ABB RobotStudio station: Estacion2.rsstn

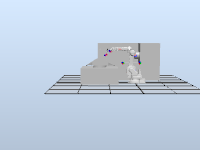
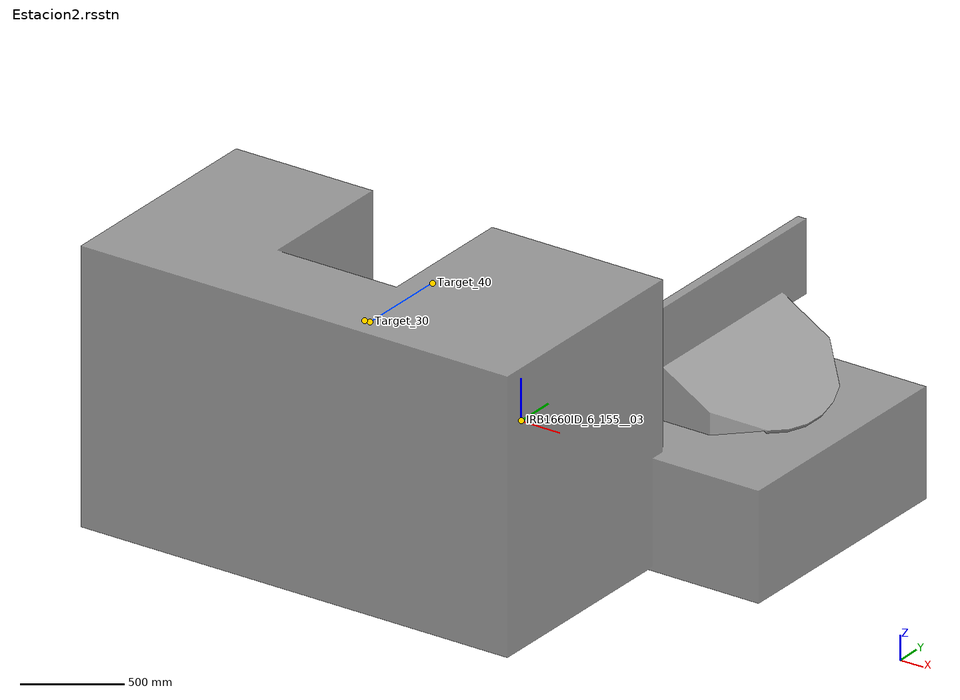
[picture v1: parts stored in the station drawn from their meshes, with robot base, taught points and paths (robot models come from the ABB library and are not in the file)]
Station Estacion2 (saved by RobotStudio 21.2.9526.0)
Controller Controlador7
  mechanical unit ROB_1: IRB1660ID_6_155__03, 6 joints, base frame (0, 0, 0) mm
Layout (positions relative to the parent item):
  - IRB1660ID_6_155__03 [mechanism, from Robots\IRB1660ID_6_155__03.rslib] at (0, 0, 0) mm; joint values [0, 0, 0, 0, 0.5236, 0] (rad or m)
  - Torno [part] at (-1068.13, -2159.82, 1500) mm, size 2500 x 1300 x 1500 mm
  - MyTool [mechanism, from Training Objects\myTool.rslib] at (944.87, 0, 1229) mm, rotated rx 180 ry 60 rz 180 deg
  - Conjunto_para_piezas_2 [part] at (775.61, 1355.8, 432.1) mm, rotated rx 90 ry 0 rz 0 deg, size 1400 x 1300 x 1400 mm
Attachment: MyTool is attached to IRB1660ID_6_155__03 / Link6
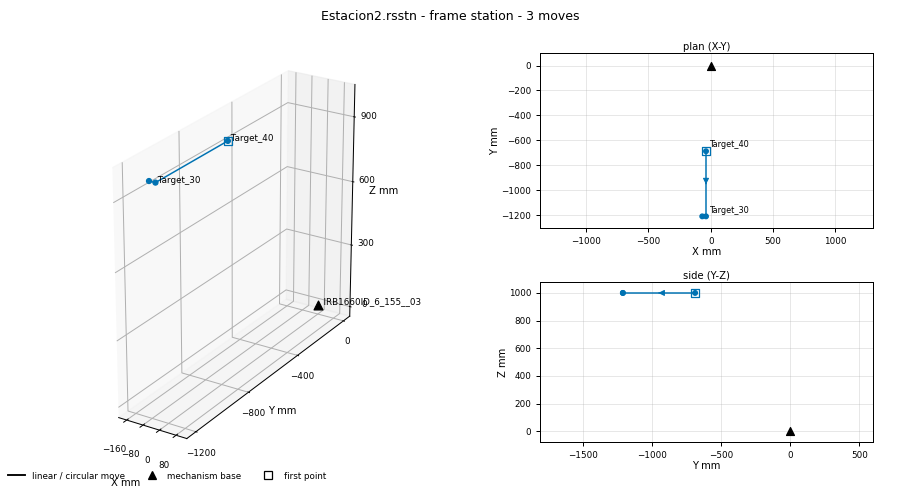
[picture p0: tool path of Estacion2.rsstn in frame station, 3 of 3 moves have a stored position in this frame; points joined in program order, loops and branches not executed]
Targets, tools, work objects and paths stored in the station, written as RAPID:
! task T_ROB1
MODULE CalibData
  TASK PERS wobjdata Workobject_1:=[FALSE,TRUE,"",[[-268.126,-859.82,700],[0.930866899,-0.099519219,0.191708757,0.294670143]],[[526.984,-410.728,208.782],[0.923994843,-0.066344622,0.1461728,0.347081306]]];
  PERS tooldata MyTool:=[TRUE,[[31.792631019,0,229.638935148],[0.945518576,0,0.325568154,0]],[1,[0,0,1],[1,0,0,0],0,0,0]];
ENDMODULE

! task T_ROB1
MODULE Module1
  CONST robtarget Target_20:=[[-499.358490679,440.828818178,-137.152602332],[0.279321138,-0.327591641,-0.74346151,-0.511789411],[-1,-1,-1,0],[9E+09,9E+09,9E+09,9E+09,9E+09,9E+09]];
  CONST robtarget Target_30:=[[-496.95439097,412.464573248,-127.534514763],[0.279321197,-0.327591644,-0.743461476,-0.511789426],[-1,-1,-1,0],[9E+09,9E+09,9E+09,9E+09,9E+09,9E+09]];
  CONST robtarget Target_40:=[[-93.00179854,549.122328966,174.503291077],[0.279321174,-0.327591615,-0.743461484,-0.511789446],[-1,-1,-1,0],[9E+09,9E+09,9E+09,9E+09,9E+09,9E+09]];
  CONST robtarget Target_50:=[[477.009747784,-354.356467387,1009.981583526],[0.460163129,0.607479572,0.647306118,0.014603227],[0,0,0,0],[9E+09,9E+09,9E+09,9E+09,9E+09,9E+09]];
  PROC Path_10()
    MoveJ Target_40,v400,z100,MyTool\WObj:=Workobject_1;
    MoveL Target_30,v200,z100,MyTool\WObj:=Workobject_1;
    MoveL Target_20,v200,z100,MyTool\WObj:=Workobject_1;
  ENDPROC
ENDMODULE

